{attribute addProperty BoxType "EL6201-0000-0017"}
{attribute addProperty Id "Slave_25A_DO0BIT10.125193Slave_25A_DO1BIT10.125194Slave_25A_DO2BIT10.125195Slave_25A_DO3BIT10.125196Slave_25B_DO0BIT10.125197Slave_25B_DO1BIT10.125198Slave_25B_DO2BIT10.125199Slave_25B_DO3BIT10.125200"}
{attribute addProperty CRC "1839693356"}
{attribute addProperty SizeInBites "8"}
{attribute addProperty SizeInBytes "1"}
TYPE Slave_25_Outputs_6DA77E2C :
STRUCT
	{attribute addProperty Name "Slave_25A_DO0"}
	Slave_25A_DO0 : BIT;
	{attribute addProperty Name "Slave_25A_DO1"}
	Slave_25A_DO1 : BIT;
	{attribute addProperty Name "Slave_25A_DO2"}
	Slave_25A_DO2 : BIT;
	{attribute addProperty Name "Slave_25A_DO3"}
	Slave_25A_DO3 : BIT;
	{attribute addProperty Name "Slave_25B_DO0"}
	Slave_25B_DO0 : BIT;
	{attribute addProperty Name "Slave_25B_DO1"}
	Slave_25B_DO1 : BIT;
	{attribute addProperty Name "Slave_25B_DO2"}
	Slave_25B_DO2 : BIT;
	{attribute addProperty Name "Slave_25B_DO3"}
	Slave_25B_DO3 : BIT;
END_STRUCT
END_TYPE

(* stored: Version 1.2.0.0, ProductVersion 3.1.4024.9
   DUT Slave_25_Outputs_6DA77E2C: Id {d338af7b-e69e-4b44-a4c1-e0ef52b18905} *)
